FUNCTION_BLOCK FB_Mb_TestGood EXTENDS FB_ModbusDevice
VAR_INPUT
	// Holding registers: 40001..40004 contiguous, 40010 within gap 8 -> one block
	Hr1    : ST_MbPoint := (nAddr := 40001);
	Hr2    : ST_MbPoint := (nAddr := 40002, eType := E_MbType.Int16, fRawMin := 0, fRawMax := 1000, fEngMin := 0, fEngMax := 100);
	Hr3    : ST_MbPoint := (nAddr := 40003, eType := E_MbType.Real32);
	Hr4    : ST_MbPoint := (nAddr := 40010, eType := E_MbType.UInt32);
	// Gap > 8 -> second block
	Hr5    : ST_MbPoint := (nAddr := 40100, eType := E_MbType.Text, nRegs := 8);
	// Slow -> its own block
	Hr6    : ST_MbPoint := (nAddr := 40116, ePoll := E_MbPoll.Slow);
	// Off -> no block
	Hr7    : ST_MbPoint := (nAddr := 40200, ePoll := E_MbPoll.Off);
	// Far away -> third fast HR block
	Hr8    : ST_MbPoint := (nAddr := 40400);
	Hr9    : ST_MbPoint := (nAddr := 40410);
	Hr10   : ST_MbPoint := (nAddr := 40420);
	Status : ST_MbPoint := (nAddr := 40300, eType := E_MbType.RegisterBit, nBit := 3);
	// Input registers, contiguous -> one block
	Ir1    : ST_MbPoint := (nAddr := 30001, eType := E_MbType.Real32);
	Ir2    : ST_MbPoint := (nAddr := 30003, eType := E_MbType.UInt32);
	// Coils and a discrete input
	Coil1  : ST_MbPoint := (nAddr := 1);
	Coil2  : ST_MbPoint := (nAddr := 2);
	Di1    : ST_MbPoint := (nAddr := 10001);
END_VAR

Register();
SUPER^();

//FB_Init is always available implicitly and it is used primarily for initialization.
//The return value is not evaluated. For a specific influence, you can also declare the
//methods explicitly and provide additional code there with the standard initialization
//code. You can evaluate the return value.
METHOD FB_Init: BOOL
VAR_INPUT
    bInitRetains: BOOL; // TRUE: the retain variables are initialized (reset warm / reset cold)
    bInCopyCode: BOOL;  // TRUE: the instance will be copied to the copy code afterward (online change)   
END_VAR
Register();
END_METHOD

METHOD FB_Reinit: BOOL
VAR_INPUT   
END_VAR
Register();
END_METHOD

METHOD PRIVATE Register
Profile(sModel := 'TestGood', eWordOrder := E_MbWordOrder.CDAB);
AddPoint(Hr1, 'Hr1');
AddPoint(Hr2, 'Hr2');
AddPoint(Hr3, 'Hr3');
AddPoint(Hr4, 'Hr4');
AddPoint(Hr5, 'Hr5');
AddPoint(Hr6, 'Hr6');
AddPoint(Hr7, 'Hr7');
AddPoint(Hr8, 'Hr8');
AddPoint(Hr9, 'Hr9');
AddPoint(Hr10, 'Hr10');
AddPoint(Status, 'Status');
AddPoint(Ir1, 'Ir1');
AddPoint(Ir2, 'Ir2');
AddPoint(Coil1, 'Coil1');
AddPoint(Coil2, 'Coil2');
AddPoint(Di1, 'Di1');
END_METHOD

END_FUNCTION_BLOCK

(* stored: Version 1.1.0.1
   POU FB_Mb_TestGood: Id {e4d0eb77-8355-4b40-946d-991f3fb665a3}, SpecialFunc None
   Method FB_Init: Id {5a2f40d8-8abf-459d-8add-8082e693055e}
   Method FB_Reinit: Id {0c898509-e052-4d6a-8fb1-74933b0af58b}
   Method Register: Id {e78f7ea8-d630-45b5-a953-095abdbf870e} *)
